// TIA Portal V18 export
FUNCTION_BLOCK "_ML2_target_supplier"   // FB29, FBD
{ S7_Optimized_Access := 'TRUE' }
VERSION : 0.1
// stored: AutoNumber true, IsIECCheckEnabled false, IsRetainMemResEnabled false, MemoryReserve 100, SetENOAutomatically false, UDAEnableTagReadback false
   VAR_INPUT
      ALLOWED : Bool;
      xServiceKey : Bool;
      xManButtonAny : Bool;
      xSwAutoCycle : Bool;
      xXrayCycleRuning : Bool;
      xGoToNextDefect : Bool;
      xGoToPrevDefect : Bool;
      xHome : Bool;
      xLoad : Bool;
      xControl1 : Bool;
      xControl2 : Bool;
      xDefectSave : Bool;
      xDefectsReset : Bool;
      Spots_pos_AR : "typeSpotList";
      CurPositios : "typePositions";
      ACK : Bool;
      ArrivedAll : Bool;
      HomePos : "typePositions";
      LoadPos : "typePositions";
      Control1Pos : "typePositions";
      Control2Pos : "typePositions";
      bSoftStop : Bool;
   END_VAR
   VAR_OUTPUT
      ExecuteAllAxisTogether : Bool;
      mdNotAllowed : Bool;
      mdServiceKey : Bool;
      mdCycle : Bool;
      mdSemi : Bool;
      mdMan : Bool;
      wsMODE : WString;
      wsTarget : WString;
      er_ws : WString;
   END_VAR
   VAR_IN_OUT
      Target_pos : "typePositions";
      DefectsDB : "typeDefectsDB";
      hmiGoToDefect : Bool;
      hmiGotoSpot : Bool;
      SPOT_i : Int;
      xyBeepDoneDefects : Bool;
   END_VAR
   VAR
      def_util_db { S7_SetPoint := 'True'} : "defects_util";
      mdSemi_was : Bool;
      st_goToDefectNow : Bool;
      q0_auto : Bool;
      q00_semi : Bool;
      q1_spot : Bool;
      p1_spot : Bool;
      q2_defect : Bool;
      p2_defect : Bool;
      q99_none : Bool;
      q_auto_waiting : Bool;
      block1 { S7_SetPoint := 'True'} : "_ML2_ts_block1";
      p3_home : Bool;
      q3_home : Bool;
      p4_load : Bool;
      q4_load : Bool;
      p5_control1 : Bool;
      q5_control1 : Bool;
      p6_control2 : Bool;
      q6_control2 : Bool;
   END_VAR
   VAR_TEMP
      locSpot_i_winBounds : Bool;
      locDefect_i_winBounds : Bool;
   END_VAR
   VAR CONSTANT
      wm_not_allowed : WString := WSTRING#'Авария';
      wm_cycle : WString := WSTRING#'Автомат';
      wm_service_key : WString := WSTRING#'Сервисный Режим';
      wm_semi_auto : WString := WSTRING#'Полуавтомат';
      wm_man : WString := WSTRING#'Ручной';
      wt00_off : WString := WSTRING#'цель не задана';
      wt0_cycle : WString := WSTRING#'автомат к точке';
      wt1_spot_man : WString := WSTRING#'ручной к точке';
      wt2_defect : WString := WSTRING#'к дефекту';
      wt3_Home : WString := WSTRING#'к домашней позиции';
      wt4_load : WString := WSTRING#'к позиции загрузки';
      wt5_Control1 : WString := WSTRING#'к первому шву';
      wt6_Control2 : WString := WSTRING#'ко второму шву';
      erws_spot_i_lt0_gt_n : WString := WSTRING#'erws_spot_i_lt0_gt_n';
      erws_defect_i_lt0_gt_n_1 : WString := WSTRING#'erws_defecti_lt0_gt_n';
   END_VAR
   VAR_TEMP   // added for the SCL form of the ladder/FBD networks
      _w1 : Bool;
   END_VAR
BEGIN

REGION Network 1
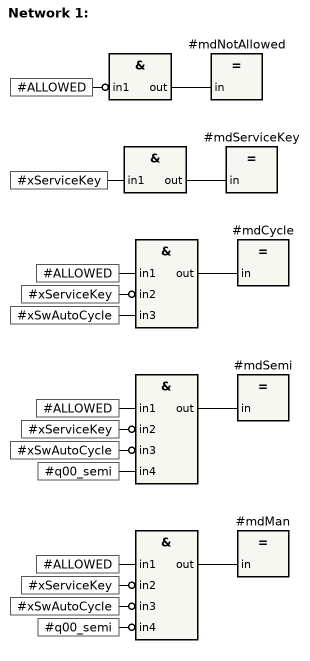
   #mdNotAllowed := NOT #ALLOWED;
   #mdServiceKey := #xServiceKey;
   #mdCycle := #ALLOWED AND NOT #xServiceKey AND #xSwAutoCycle;
   #mdSemi := #ALLOWED AND NOT #xServiceKey AND NOT #xSwAutoCycle AND #q00_semi;
   #mdMan := #ALLOWED AND NOT #xServiceKey AND NOT #xSwAutoCycle AND NOT #q00_semi;
END_REGION

REGION Network 2
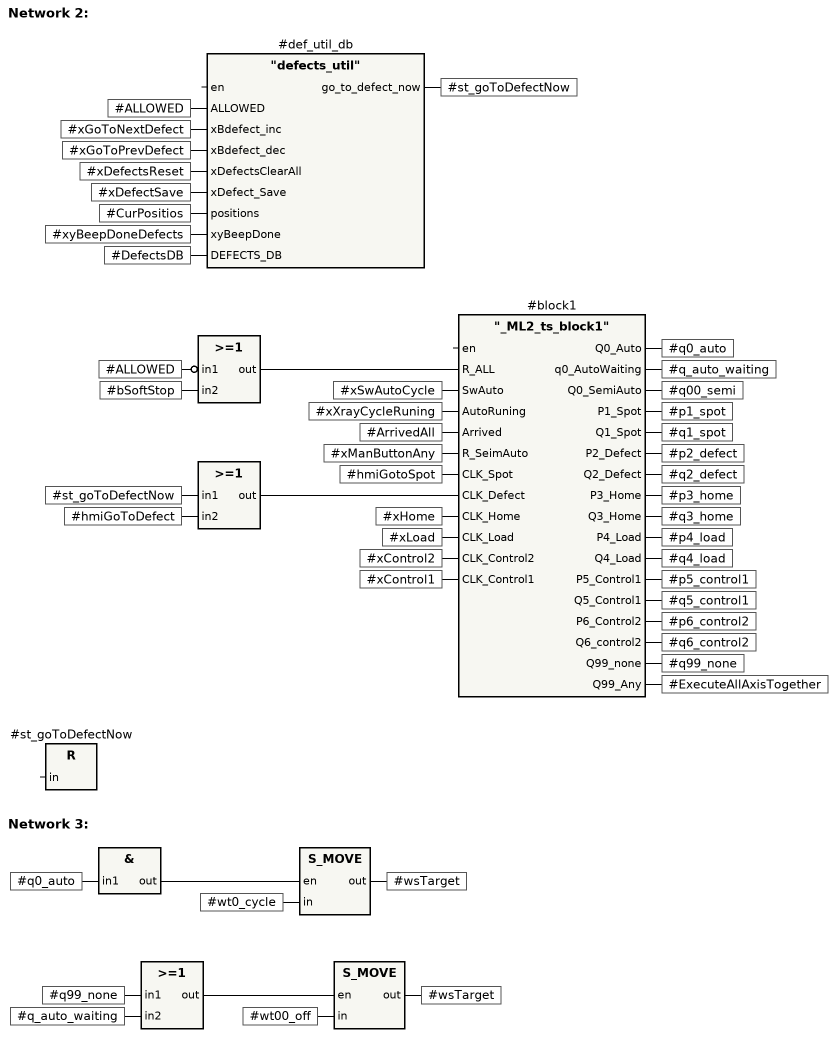
   #def_util_db(ALLOWED := #ALLOWED,   // "defects_util"
                xBdefect_inc := #xGoToNextDefect,
                xBdefect_dec := #xGoToPrevDefect,
                xDefectsClearAll := #xDefectsReset,
                xDefect_Save := #xDefectSave,
                positions := #CurPositios,
                xyBeepDone := #xyBeepDoneDefects,
                DEFECTS_DB := #DefectsDB,
                go_to_defect_now => #st_goToDefectNow);
   #block1(R_ALL := NOT #ALLOWED OR #bSoftStop,   // "_ML2_ts_block1"
           SwAuto := #xSwAutoCycle,
           AutoRuning := #xXrayCycleRuning,
           Arrived := #ArrivedAll,
           R_SeimAuto := #xManButtonAny,
           CLK_Spot := #hmiGotoSpot,
           CLK_Defect := #st_goToDefectNow OR #hmiGoToDefect,
           CLK_Home := #xHome,
           CLK_Load := #xLoad,
           CLK_Control2 := #xControl2,
           CLK_Control1 := #xControl1,
           Q0_Auto => #q0_auto,
           q0_AutoWaiting => #q_auto_waiting,
           Q0_SemiAuto => #q00_semi,
           P1_Spot => #p1_spot,
           Q1_Spot => #q1_spot,
           P2_Defect => #p2_defect,
           Q2_Defect => #q2_defect,
           P3_Home => #p3_home,
           Q3_Home => #q3_home,
           P4_Load => #p4_load,
           Q4_Load => #q4_load,
           P5_Control1 => #p5_control1,
           Q5_Control1 => #q5_control1,
           P6_Control2 => #p6_control2,
           Q6_control2 => #q6_control2,
           Q99_none => #q99_none,
           Q99_Any => #ExecuteAllAxisTogether);
   #st_goToDefectNow := FALSE;
END_REGION

REGION Network 3
   IF #q0_auto THEN #wsTarget := #wt0_cycle; END_IF;
   IF #q99_none OR #q_auto_waiting THEN #wsTarget := #wt00_off; END_IF;
END_REGION

REGION Network 4
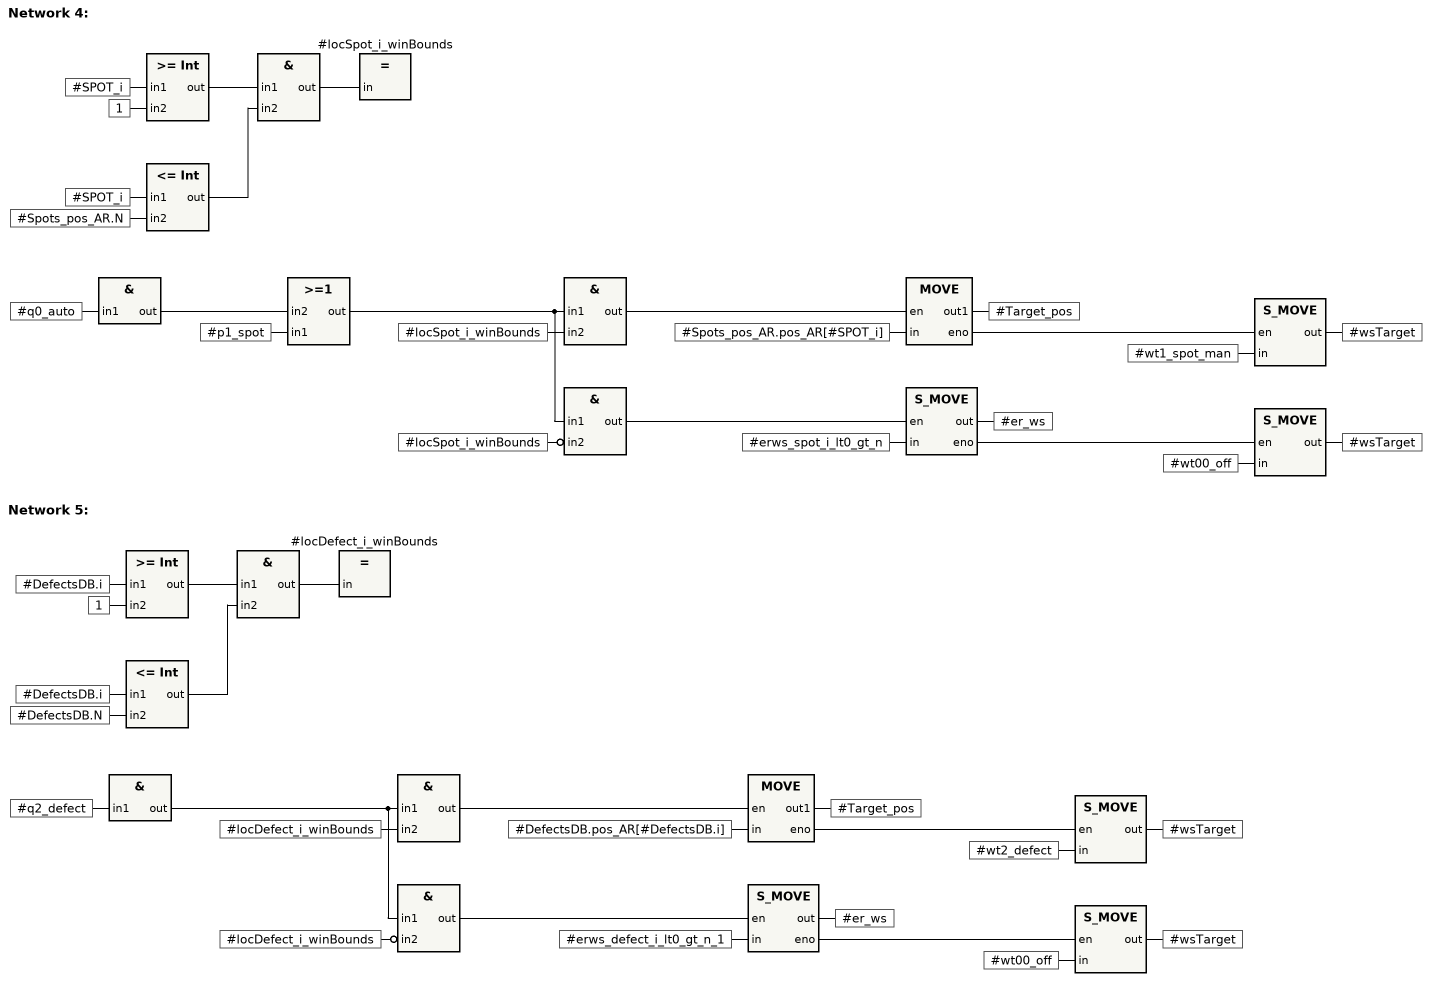
   #locSpot_i_winBounds := (#SPOT_i >= 1) AND (#SPOT_i <= #Spots_pos_AR.N);
   #_w1 := #q0_auto OR #p1_spot;
   IF #_w1 AND #locSpot_i_winBounds THEN
       #Target_pos := #Spots_pos_AR.pos_AR[#SPOT_i];
       #wsTarget := #wt1_spot_man;
   END_IF;
   IF #_w1 AND NOT #locSpot_i_winBounds THEN
       #er_ws := #erws_spot_i_lt0_gt_n;
       #wsTarget := #wt00_off;
   END_IF;
END_REGION

REGION Network 5
   #locDefect_i_winBounds := (#DefectsDB.i >= 1) AND (#DefectsDB.i <= #DefectsDB.N);
   IF #q2_defect AND #locDefect_i_winBounds THEN
       #Target_pos := #DefectsDB.pos_AR[#DefectsDB.i];
       #wsTarget := #wt2_defect;
   END_IF;
   IF #q2_defect AND NOT #locDefect_i_winBounds THEN
       #er_ws := #erws_defect_i_lt0_gt_n_1;
       #wsTarget := #wt00_off;
   END_IF;
END_REGION

REGION Network 6
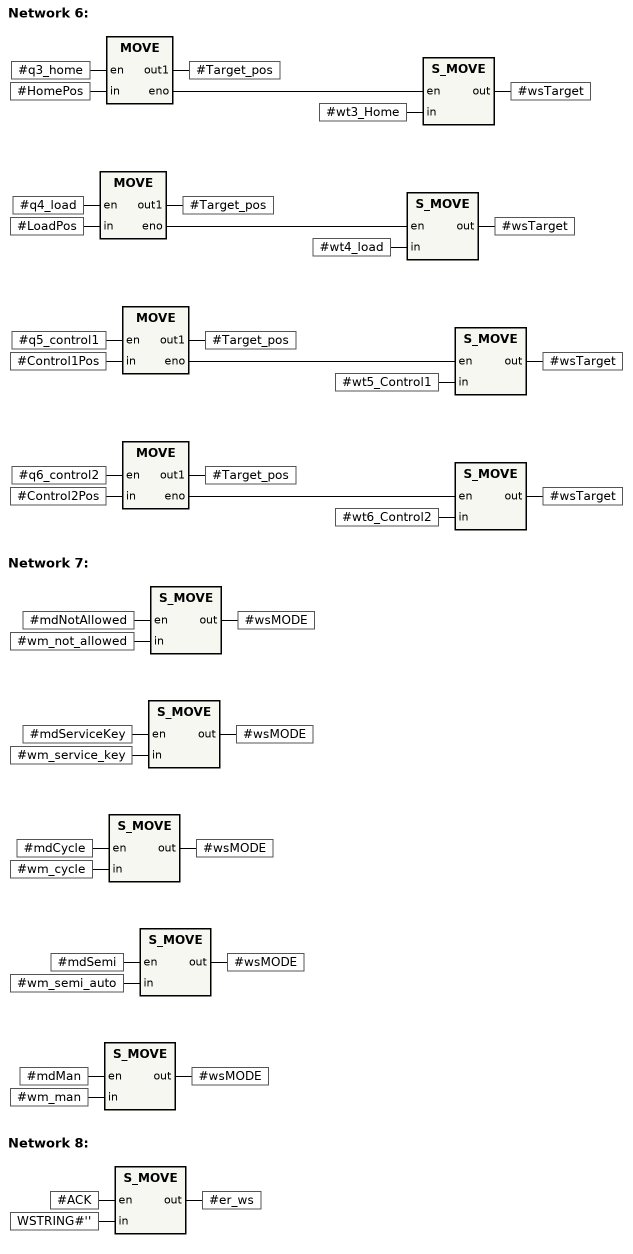
   IF #q3_home THEN
       #Target_pos := #HomePos;
       #wsTarget := #wt3_Home;
   END_IF;
   IF #q4_load THEN
       #Target_pos := #LoadPos;
       #wsTarget := #wt4_load;
   END_IF;
   IF #q5_control1 THEN
       #Target_pos := #Control1Pos;
       #wsTarget := #wt5_Control1;
   END_IF;
   IF #q6_control2 THEN
       #Target_pos := #Control2Pos;
       #wsTarget := #wt6_Control2;
   END_IF;
END_REGION

REGION Network 7
   IF #mdNotAllowed THEN #wsMODE := #wm_not_allowed; END_IF;
   IF #mdServiceKey THEN #wsMODE := #wm_service_key; END_IF;
   IF #mdCycle THEN #wsMODE := #wm_cycle; END_IF;
   IF #mdSemi THEN #wsMODE := #wm_semi_auto; END_IF;
   IF #mdMan THEN #wsMODE := #wm_man; END_IF;
END_REGION

REGION Network 8
   IF #ACK THEN #er_ws := WSTRING#''; END_IF;
END_REGION
END_FUNCTION_BLOCK
